Staubli VAL3: io.pjx

--- io.pjx ---
Parameters version=s7.9.1 stackSize=0 millimeterUnit=true
Data file=io.dtx

--- io.dtx ---
public sio IOC = {link=Socket\MFX}
